TEXTLIST TextList_Pompage
  0 = 'Pomp inter' | FR: 'Pompage interjoints' | EN: 'Inter ring pumping'
  1 = 'Confirm regen' | FR: 'Confirmer régénération ?' | EN: 'Confirm regeneration ?'
   = ''
END_TEXTLIST

(* stored: Version 1.1.0.1, ProductVersion 3.1.4024.10
   TextList TextList_Pompage: Id {f8749c8a-19a7-40eb-9223-96489266e293} *)
